  movej([1.2951, -1.388, 1.6, -0.4, 1.57, 0.0], a=1.7, v=2.0, r=0.08)
  movej([1.2954, -1.3912, 1.6, -0.4, 1.57, 0.0], a=1.7, v=2.0, r=0.08)
  movej([1.2958, -1.3945, 1.6, -0.4, 1.57, 0.0], a=1.7, v=2.0, r=0.08)
  movej([1.2961, -1.3977, 1.6, -0.4, 1.57, 0.0], a=1.7, v=2.0, r=0.08)
  movej([1.2965, -1.4009, 1.6, -0.4, 1.57, 0.0], a=1.7, v=2.0, r=0.08)
  movej([1.2969, -1.4041, 1.6, -0.4, 1.57, 0.0], a=1.7, v=2.0, r=0.08)
  movej([1.2973, -1.4072, 1.6, -0.4, 1.57, 0.0], a=1.7, v=2.0, r=0.08)
  movej([1.2977, -1.4104, 1.6, -0.4, 1.57, 0.0], a=1.7, v=2.0, r=0.08)
  movej([1.2982, -1.4135, 1.6, -0.4, 1.57, 0.0], a=1.7, v=2.0, r=0.08)
  movej([1.2986, -1.4166, 1.6, -0.4, 1.57, 0.0], a=1.7, v=2.0, r=0.08)
  movej([1.2991, -1.4196, 1.6, -0.4, 1.57, 0.0], a=1.7, v=2.0, r=0.08)
  movej([1.2996, -1.4227, 1.6, -0.4, 1.57, 0.0], a=1.7, v=2.0, r=0.08)
  movej([1.3001, -1.4257, 1.6, -0.4, 1.57, 0.0], a=1.7, v=2.0, r=0.08)
  movej([1.3006, -1.4287, 1.6, -0.4, 1.57, 0.0], a=1.7, v=2.0, r=0.08)
  movej([1.3012, -1.4317, 1.6, -0.4, 1.57, 0.0], a=1.7, v=2.0, r=0.08)
  movej([1.3018, -1.4347, 1.6, -0.4, 1.57, 0.0], a=1.7, v=2.0, r=0.08)
  movej([1.3023, -1.4376, 1.6, -0.4, 1.57, 0.0], a=1.7, v=2.0, r=0.08)
  movej([1.3029, -1.4405, 1.6, -0.4, 1.57, 0.0], a=1.7, v=2.0, r=0.08)
  movej([1.3035, -1.4433, 1.6, -0.4, 1.57, 0.0], a=1.7, v=2.0, r=0.08)
  movej([1.3042, -1.4462, 1.6, -0.4, 1.57, 0.0], a=1.7, v=2.0, r=0.08)
  movej([1.3048, -1.449, 1.6, -0.4, 1.57, 0.0], a=1.7, v=2.0, r=0.08)
  movej([1.3055, -1.4518, 1.6, -0.4, 1.57, 0.0], a=1.7, v=2.0, r=0.08)
  movej([1.3061, -1.4545, 1.6, -0.4, 1.57, 0.0], a=1.7, v=2.0, r=0.08)
  movej([1.3068, -1.4572, 1.6, -0.4, 1.57, 0.0], a=1.7, v=2.0, r=0.08)
  movej([1.3075, -1.4599, 1.6, -0.4, 1.57, 0.0], a=1.7, v=2.0, r=0.08)
  movej([1.3083, -1.4626, 1.6, -0.4, 1.57, 0.0], a=1.7, v=2.0, r=0.08)
  movej([1.309, -1.4652, 1.6, -0.4, 1.57, 0.0], a=1.7, v=2.0, r=0.08)
  movej([1.3098, -1.4678, 1.6, -0.4, 1.57, 0.0], a=1.7, v=2.0, r=0.08)
  movej([1.3105, -1.4703, 1.6, -0.4, 1.57, 0.0], a=1.7, v=2.0, r=0.08)
  movej([1.3113, -1.4728, 1.6, -0.4, 1.57, 0.0], a=1.7, v=2.0, r=0.08)
  movej([1.3121, -1.4753, 1.6, -0.4, 1.57, 0.0], a=1.7, v=2.0, r=0.08)
  movej([1.313, -1.4777, 1.6, -0.4, 1.57, 0.0], a=1.7, v=2.0, r=0.08)
  movej([1.3138, -1.4801, 1.6, -0.4, 1.57, 0.0], a=1.7, v=2.0, r=0.08)
  movej([1.3146, -1.4825, 1.6, -0.4, 1.57, 0.0], a=1.7, v=2.0, r=0.08)
  movej([1.3155, -1.4848, 1.6, -0.4, 1.57, 0.0], a=1.7, v=2.0, r=0.08)
  movej([1.3164, -1.4871, 1.6, -0.4, 1.57, 0.0], a=1.7, v=2.0, r=0.08)
  movej([1.3173, -1.4894, 1.6, -0.4, 1.57, 0.0], a=1.7, v=2.0, r=0.08)
  movej([1.3182, -1.4916, 1.6, -0.4, 1.57, 0.0], a=1.7, v=2.0, r=0.08)
  movej([1.3191, -1.4937, 1.6, -0.4, 1.57, 0.0], a=1.7, v=2.0, r=0.08)
  movej([1.3201, -1.4959, 1.6, -0.4, 1.57, 0.0], a=1.7, v=2.0, r=0.08)
  movej([1.321, -1.4979, 1.6, -0.4, 1.57, 0.0], a=1.7, v=2.0, r=0.08)
  movej([1.322, -1.5, 1.6, -0.4, 1.57, 0.0], a=1.7, v=2.0, r=0.08)
  movej([1.323, -1.502, 1.6, -0.4, 1.57, 0.0], a=1.7, v=2.0, r=0.08)
  movej([1.324, -1.5039, 1.6, -0.4, 1.57, 0.0], a=1.7, v=2.0, r=0.08)
  movej([1.3251, -1.5058, 1.6, -0.4, 1.57, 0.0], a=1.7, v=2.0, r=0.08)
  movej([1.3261, -1.5077, 1.6, -0.4, 1.57, 0.0], a=1.7, v=2.0, r=0.08)
  movej([1.3271, -1.5095, 1.6, -0.4, 1.57, 0.0], a=1.7, v=2.0, r=0.08)
  movej([1.3282, -1.5113, 1.6, -0.4, 1.57, 0.0], a=1.7, v=2.0, r=0.08)
  movej([1.3293, -1.513, 1.6, -0.4, 1.57, 0.0], a=1.7, v=2.0, r=0.08)
  movej([1.3304, -1.5147, 1.6, -0.4, 1.57, 0.0], a=1.7, v=2.0, r=0.08)
  movej([1.3315, -1.5163, 1.6, -0.4, 1.57, 0.0], a=1.7, v=2.0, r=0.08)
  movej([1.3326, -1.5179, 1.6, -0.4, 1.57, 0.0], a=1.7, v=2.0, r=0.08)
  movej([1.3338, -1.5194, 1.6, -0.4, 1.57, 0.0], a=1.7, v=2.0, r=0.08)
  movej([1.3349, -1.5209, 1.6, -0.4, 1.57, 0.0], a=1.7, v=2.0, r=0.08)
  movej([1.3361, -1.5224, 1.6, -0.4, 1.57, 0.0], a=1.7, v=2.0, r=0.08)
  movej([1.3373, -1.5238, 1.6, -0.4, 1.57, 0.0], a=1.7, v=2.0, r=0.08)
  movej([1.3385, -1.5251, 1.6, -0.4, 1.57, 0.0], a=1.7, v=2.0, r=0.08)
  movej([1.3397, -1.5264, 1.6, -0.4, 1.57, 0.0], a=1.7, v=2.0, r=0.08)
  movej([1.3409, -1.5277, 1.6, -0.4, 1.57, 0.0], a=1.7, v=2.0, r=0.08)
  movej([1.3422, -1.5288, 1.6, -0.4, 1.57, 0.0], a=1.7, v=2.0, r=0.08)
  movej([1.3434, -1.53, 1.6, -0.4, 1.57, 0.0], a=1.7, v=2.0, r=0.08)
  movej([1.3447, -1.5311, 1.6, -0.4, 1.57, 0.0], a=1.7, v=2.0, r=0.08)
  movej([1.346, -1.5321, 1.6, -0.4, 1.57, 0.0], a=1.7, v=2.0, r=0.08)
  movej([1.3473, -1.5331, 1.6, -0.4, 1.57, 0.0], a=1.7, v=2.0, r=0.08)
  movej([1.3486, -1.5341, 1.6, -0.4, 1.57, 0.0], a=1.7, v=2.0, r=0.08)
  movej([1.3499, -1.535, 1.6, -0.4, 1.57, 0.0], a=1.7, v=2.0, r=0.08)
  movej([1.3513, -1.5358, 1.6, -0.4, 1.57, 0.0], a=1.7, v=2.0, r=0.08)
  movej([1.3526, -1.5366, 1.6, -0.4, 1.57, 0.0], a=1.7, v=2.0, r=0.08)
  movej([1.354, -1.5373, 1.6, -0.4, 1.57, 0.0], a=1.7, v=2.0, r=0.08)
  movej([1.3554, -1.538, 1.6, -0.4, 1.57, 0.0], a=1.7, v=2.0, r=0.08)
  movej([1.3568, -1.5386, 1.6, -0.4, 1.57, 0.0], a=1.7, v=2.0, r=0.08)
  movej([1.3582, -1.5392, 1.6, -0.4, 1.57, 0.0], a=1.7, v=2.0, r=0.08)
  movej([1.3596, -1.5397, 1.6, -0.4, 1.57, 0.0], a=1.7, v=2.0, r=0.08)
  movej([1.361, -1.5402, 1.6, -0.4, 1.57, 0.0], a=1.7, v=2.0, r=0.08)
  movej([1.3625, -1.5406, 1.6, -0.4, 1.57, 0.0], a=1.7, v=2.0, r=0.08)
  movej([1.3639, -1.541, 1.6, -0.4, 1.57, 0.0], a=1.7, v=2.0, r=0.08)
  movej([1.3654, -1.5413, 1.6, -0.4, 1.57, 0.0], a=1.7, v=2.0, r=0.08)
  movej([1.3669, -1.5416, 1.6, -0.4, 1.57, 0.0], a=1.7, v=2.0, r=0.08)
  movej([1.3684, -1.5418, 1.6, -0.4, 1.57, 0.0], a=1.7, v=2.0, r=0.08)
  movej([1.3699, -1.5419, 1.6, -0.4, 1.57, 0.0], a=1.7, v=2.0, r=0.08)
  movej([1.3714, -1.542, 1.6, -0.4, 1.57, 0.0], a=1.7, v=2.0, r=0.08)
  movej([1.373, -1.5421, 1.6, -0.4, 1.57, 0.0], a=1.7, v=2.0, r=0.08)
  movej([1.3745, -1.5421, 1.6, -0.4, 1.57, 0.0], a=1.7, v=2.0, r=0.08)
  movej([1.3761, -1.542, 1.6, -0.4, 1.57, 0.0], a=1.7, v=2.0, r=0.08)
  movej([1.3776, -1.5419, 1.6, -0.4, 1.57, 0.0], a=1.7, v=2.0, r=0.08)
  movej([1.3792, -1.5417, 1.6, -0.4, 1.57, 0.0], a=1.7, v=2.0, r=0.08)
  movej([1.3808, -1.5415, 1.6, -0.4, 1.57, 0.0], a=1.7, v=2.0, r=0.08)
  movej([1.3824, -1.5412, 1.6, -0.4, 1.57, 0.0], a=1.7, v=2.0, r=0.08)
  movej([1.384, -1.5409, 1.6, -0.4, 1.57, 0.0], a=1.7, v=2.0, r=0.08)
  movej([1.3857, -1.5405, 1.6, -0.4, 1.57, 0.0], a=1.7, v=2.0, r=0.08)
  movej([1.3873, -1.5401, 1.6, -0.4, 1.57, 0.0], a=1.7, v=2.0, r=0.08)
  movej([1.389, -1.5396, 1.6, -0.4, 1.57, 0.0], a=1.7, v=2.0, r=0.08)
  movej([1.3906, -1.5391, 1.6, -0.4, 1.57, 0.0], a=1.7, v=2.0, r=0.08)
  movej([1.3923, -1.5385, 1.6, -0.4, 1.57, 0.0], a=1.7, v=2.0, r=0.08)
  movej([1.394, -1.5378, 1.6, -0.4, 1.57, 0.0], a=1.7, v=2.0, r=0.08)
  movej([1.3957, -1.5371, 1.6, -0.4, 1.57, 0.0], a=1.7, v=2.0, r=0.08)
  movej([1.3974, -1.5364, 1.6, -0.4, 1.57, 0.0], a=1.7, v=2.0, r=0.08)
  movej([1.3991, -1.5356, 1.6, -0.4, 1.57, 0.0], a=1.7, v=2.0, r=0.08)
  movej([1.4008, -1.5347, 1.6, -0.4, 1.57, 0.0], a=1.7, v=2.0, r=0.08)
  movej([1.4026, -1.5338, 1.6, -0.4, 1.57, 0.0], a=1.7, v=2.0, r=0.08)
  movej([1.4043, -1.5329, 1.6, -0.4, 1.57, 0.0], a=1.7, v=2.0, r=0.08)
  movej([1.4061, -1.5319, 1.6, -0.4, 1.57, 0.0], a=1.7, v=2.0, r=0.08)
  movej([1.4078, -1.5308, 1.6, -0.4, 1.57, 0.0], a=1.7, v=2.0, r=0.08)
  movej([1.4096, -1.5297, 1.6, -0.4, 1.57, 0.0], a=1.7, v=2.0, r=0.08)
  movej([1.4114, -1.5286, 1.6, -0.4, 1.57, 0.0], a=1.7, v=2.0, r=0.08)
  movej([1.4132, -1.5273, 1.6, -0.4, 1.57, 0.0], a=1.7, v=2.0, r=0.08)
  movej([1.415, -1.5261, 1.6, -0.4, 1.57, 0.0], a=1.7, v=2.0, r=0.08)
  movej([1.4168, -1.5248, 1.6, -0.4, 1.57, 0.0], a=1.7, v=2.0, r=0.08)
  movej([1.4187, -1.5234, 1.6, -0.4, 1.57, 0.0], a=1.7, v=2.0, r=0.08)
  movej([1.4205, -1.522, 1.6, -0.4, 1.57, 0.0], a=1.7, v=2.0, r=0.08)
  movej([1.4223, -1.5206, 1.6, -0.4, 1.57, 0.0], a=1.7, v=2.0, r=0.08)
  movej([1.4242, -1.5191, 1.6, -0.4, 1.57, 0.0], a=1.7, v=2.0, r=0.08)
  movej([1.4261, -1.5175, 1.6, -0.4, 1.57, 0.0], a=1.7, v=2.0, r=0.08)
  movej([1.4279, -1.5159, 1.6, -0.4, 1.57, 0.0], a=1.7, v=2.0, r=0.08)
  movej([1.4298, -1.5143, 1.6, -0.4, 1.57, 0.0], a=1.7, v=2.0, r=0.08)
  movej([1.4317, -1.5126, 1.6, -0.4, 1.57, 0.0], a=1.7, v=2.0, r=0.08)
  movej([1.4336, -1.5108, 1.6, -0.4, 1.57, 0.0], a=1.7, v=2.0, r=0.08)
  movej([1.4355, -1.509, 1.6, -0.4, 1.57, 0.0], a=1.7, v=2.0, r=0.08)
  movej([1.4374, -1.5072, 1.6, -0.4, 1.57, 0.0], a=1.7, v=2.0, r=0.08)
  movej([1.4394, -1.5053, 1.6, -0.4, 1.57, 0.0], a=1.7, v=2.0, r=0.08)
  movej([1.4413, -1.5034, 1.6, -0.4, 1.57, 0.0], a=1.7, v=2.0, r=0.08)
  movej([1.4432, -1.5015, 1.6, -0.4, 1.57, 0.0], a=1.7, v=2.0, r=0.08)
  movej([1.4452, -1.4995, 1.6, -0.4, 1.57, 0.0], a=1.7, v=2.0, r=0.08)
  movej([1.4471, -1.4974, 1.6, -0.4, 1.57, 0.0], a=1.7, v=2.0, r=0.08)
  movej([1.4491, -1.4953, 1.6, -0.4, 1.57, 0.0], a=1.7, v=2.0, r=0.08)
  movej([1.4511, -1.4932, 1.6, -0.4, 1.57, 0.0], a=1.7, v=2.0, r=0.08)
  movej([1.453, -1.491, 1.6, -0.4, 1.57, 0.0], a=1.7, v=2.0, r=0.08)
  movej([1.455, -1.4888, 1.6, -0.4, 1.57, 0.0], a=1.7, v=2.0, r=0.08)
  movej([1.457, -1.4865, 1.6, -0.4, 1.57, 0.0], a=1.7, v=2.0, r=0.08)
  movej([1.459, -1.4843, 1.6, -0.4, 1.57, 0.0], a=1.7, v=2.0, r=0.08)
  movej([1.461, -1.4819, 1.6, -0.4, 1.57, 0.0], a=1.7, v=2.0, r=0.08)
  movej([1.463, -1.4795, 1.6, -0.4, 1.57, 0.0], a=1.7, v=2.0, r=0.08)
  movej([1.4651, -1.4771, 1.6, -0.4, 1.57, 0.0], a=1.7, v=2.0, r=0.08)
  movej([1.4671, -1.4747, 1.6, -0.4, 1.57, 0.0], a=1.7, v=2.0, r=0.08)
  movej([1.4691, -1.4722, 1.6, -0.4, 1.57, 0.0], a=1.7, v=2.0, r=0.08)
  movej([1.4712, -1.4697, 1.6, -0.4, 1.57, 0.0], a=1.7, v=2.0, r=0.08)
  movej([1.4732, -1.4671, 1.6, -0.4, 1.57, 0.0], a=1.7, v=2.0, r=0.08)
  movej([1.4753, -1.4645, 1.6, -0.4, 1.57, 0.0], a=1.7, v=2.0, r=0.08)
  movej([1.4773, -1.4619, 1.6, -0.4, 1.57, 0.0], a=1.7, v=2.0, r=0.08)
  movej([1.4794, -1.4593, 1.6, -0.4, 1.57, 0.0], a=1.7, v=2.0, r=0.08)
  movej([1.4814, -1.4566, 1.6, -0.4, 1.57, 0.0], a=1.7, v=2.0, r=0.08)
  movej([1.4835, -1.4538, 1.6, -0.4, 1.57, 0.0], a=1.7, v=2.0, r=0.08)
  movej([1.4856, -1.4511, 1.6, -0.4, 1.57, 0.0], a=1.7, v=2.0, r=0.08)
  movej([1.4877, -1.4483, 1.6, -0.4, 1.57, 0.0], a=1.7, v=2.0, r=0.08)
  movej([1.4898, -1.4455, 1.6, -0.4, 1.57, 0.0], a=1.7, v=2.0, r=0.08)
  movej([1.4919, -1.4426, 1.6, -0.4, 1.57, 0.0], a=1.7, v=2.0, r=0.08)
  movej([1.494, -1.4398, 1.6, -0.4, 1.57, 0.0], a=1.7, v=2.0, r=0.08)
  movej([1.4961, -1.4369, 1.6, -0.4, 1.57, 0.0], a=1.7, v=2.0, r=0.08)
  movej([1.4982, -1.4339, 1.6, -0.4, 1.57, 0.0], a=1.7, v=2.0, r=0.08)
  movej([1.5003, -1.431, 1.6, -0.4, 1.57, 0.0], a=1.7, v=2.0, r=0.08)
  movej([1.5024, -1.428, 1.6, -0.4, 1.57, 0.0], a=1.7, v=2.0, r=0.08)
  movej([1.5045, -1.425, 1.6, -0.4, 1.57, 0.0], a=1.7, v=2.0, r=0.08)
  movej([1.5067, -1.4219, 1.6, -0.4, 1.57, 0.0], a=1.7, v=2.0, r=0.08)
  movej([1.5088, -1.4189, 1.6, -0.4, 1.57, 0.0], a=1.7, v=2.0, r=0.08)
  movej([1.5109, -1.4158, 1.6, -0.4, 1.57, 0.0], a=1.7, v=2.0, r=0.08)
  movej([1.5131, -1.4127, 1.6, -0.4, 1.57, 0.0], a=1.7, v=2.0, r=0.08)
  movej([1.5152, -1.4096, 1.6, -0.4, 1.57, 0.0], a=1.7, v=2.0, r=0.08)
  movej([1.5173, -1.4064, 1.6, -0.4, 1.57, 0.0], a=1.7, v=2.0, r=0.08)
  movej([1.5195, -1.4033, 1.6, -0.4, 1.57, 0.0], a=1.7, v=2.0, r=0.08)
  movej([1.5216, -1.4001, 1.6, -0.4, 1.57, 0.0], a=1.7, v=2.0, r=0.08)
  movej([1.5238, -1.3969, 1.6, -0.4, 1.57, 0.0], a=1.7, v=2.0, r=0.08)
  movej([1.5259, -1.3937, 1.6, -0.4, 1.57, 0.0], a=1.7, v=2.0, r=0.08)
  movej([1.5281, -1.3904, 1.6, -0.4, 1.57, 0.0], a=1.7, v=2.0, r=0.08)
  movej([1.5303, -1.3872, 1.6, -0.4, 1.57, 0.0], a=1.7, v=2.0, r=0.08)
  movej([1.5324, -1.3839, 1.6, -0.4, 1.57, 0.0], a=1.7, v=2.0, r=0.08)
  movej([1.5346, -1.3806, 1.6, -0.4, 1.57, 0.0], a=1.7, v=2.0, r=0.08)
  movej([1.5368, -1.3773, 1.6, -0.4, 1.57, 0.0], a=1.7, v=2.0, r=0.08)
  movej([1.5389, -1.374, 1.6, -0.4, 1.57, 0.0], a=1.7, v=2.0, r=0.08)
  movej([1.5411, -1.3707, 1.6, -0.4, 1.57, 0.0], a=1.7, v=2.0, r=0.08)
  movej([1.5433, -1.3674, 1.6, -0.4, 1.57, 0.0], a=1.7, v=2.0, r=0.08)
  movej([1.5454, -1.364, 1.6, -0.4, 1.57, 0.0], a=1.7, v=2.0, r=0.08)
  movej([1.5476, -1.3607, 1.6, -0.4, 1.57, 0.0], a=1.7, v=2.0, r=0.08)
  movej([1.5498, -1.3573, 1.6, -0.4, 1.57, 0.0], a=1.7, v=2.0, r=0.08)
  movej([1.552, -1.354, 1.6, -0.4, 1.57, 0.0], a=1.7, v=2.0, r=0.08)
  movej([1.5542, -1.3506, 1.6, -0.4, 1.57, 0.0], a=1.7, v=2.0, r=0.08)
  movej([1.5563, -1.3472, 1.6, -0.4, 1.57, 0.0], a=1.7, v=2.0, r=0.08)
  movej([1.5585, -1.3438, 1.6, -0.4, 1.57, 0.0], a=1.7, v=2.0, r=0.08)
  movej([1.5607, -1.3404, 1.6, -0.4, 1.57, 0.0], a=1.7, v=2.0, r=0.08)
  movej([1.5629, -1.337, 1.6, -0.4, 1.57, 0.0], a=1.7, v=2.0, r=0.08)
  movej([1.5651, -1.3336, 1.6, -0.4, 1.57, 0.0], a=1.7, v=2.0, r=0.08)
  movej([1.5673, -1.3302, 1.6, -0.4, 1.57, 0.0], a=1.7, v=2.0, r=0.08)
  movej([1.5695, -1.3268, 1.6, -0.4, 1.57, 0.0], a=1.7, v=2.0, r=0.08)
  movej([1.5716, -1.3235, 1.6, -0.4, 1.57, 0.0], a=1.7, v=2.0, r=0.08)
  movej([1.5738, -1.3201, 1.6, -0.4, 1.57, 0.0], a=1.7, v=2.0, r=0.08)
  movej([1.576, -1.3167, 1.6, -0.4, 1.57, 0.0], a=1.7, v=2.0, r=0.08)
  movej([1.5782, -1.3133, 1.6, -0.4, 1.57, 0.0], a=1.7, v=2.0, r=0.08)
  movej([1.5804, -1.3099, 1.6, -0.4, 1.57, 0.0], a=1.7, v=2.0, r=0.08)
  movej([1.5826, -1.3065, 1.6, -0.4, 1.57, 0.0], a=1.7, v=2.0, r=0.08)
  movej([1.5847, -1.3031, 1.6, -0.4, 1.57, 0.0], a=1.7, v=2.0, r=0.08)
  movej([1.5869, -1.2997, 1.6, -0.4, 1.57, 0.0], a=1.7, v=2.0, r=0.08)
  movej([1.5891, -1.2964, 1.6, -0.4, 1.57, 0.0], a=1.7, v=2.0, r=0.08)
  movej([1.5913, -1.293, 1.6, -0.4, 1.57, 0.0], a=1.7, v=2.0, r=0.08)
  movej([1.5935, -1.2896, 1.6, -0.4, 1.57, 0.0], a=1.7, v=2.0, r=0.08)
  movej([1.5956, -1.2863, 1.6, -0.4, 1.57, 0.0], a=1.7, v=2.0, r=0.08)
  movej([1.5978, -1.283, 1.6, -0.4, 1.57, 0.0], a=1.7, v=2.0, r=0.08)
  movej([1.6, -1.2796, 1.6, -0.4, 1.57, 0.0], a=1.7, v=2.0, r=0.08)
  movej([1.6022, -1.2763, 1.6, -0.4, 1.57, 0.0], a=1.7, v=2.0, r=0.08)
  movej([1.6043, -1.273, 1.6, -0.4, 1.57, 0.0], a=1.7, v=2.0, r=0.08)
  movej([1.6065, -1.2697, 1.6, -0.4, 1.57, 0.0], a=1.7, v=2.0, r=0.08)
  movej([1.6087, -1.2665, 1.6, -0.4, 1.57, 0.0], a=1.7, v=2.0, r=0.08)
  movej([1.6108, -1.2632, 1.6, -0.4, 1.57, 0.0], a=1.7, v=2.0, r=0.08)
  movej([1.613, -1.26, 1.6, -0.4, 1.57, 0.0], a=1.7, v=2.0, r=0.08)
  movej([1.6151, -1.2567, 1.6, -0.4, 1.57, 0.0], a=1.7, v=2.0, r=0.08)
  movej([1.6173, -1.2535, 1.6, -0.4, 1.57, 0.0], a=1.7, v=2.0, r=0.08)
  movej([1.6194, -1.2503, 1.6, -0.4, 1.57, 0.0], a=1.7, v=2.0, r=0.08)
  movej([1.6216, -1.2471, 1.6, -0.4, 1.57, 0.0], a=1.7, v=2.0, r=0.08)
  movej([1.6237, -1.244, 1.6, -0.4, 1.57, 0.0], a=1.7, v=2.0, r=0.08)
  movej([1.6259, -1.2409, 1.6, -0.4, 1.57, 0.0], a=1.7, v=2.0, r=0.08)
  movej([1.628, -1.2377, 1.6, -0.4, 1.57, 0.0], a=1.7, v=2.0, r=0.08)
  movej([1.6301, -1.2347, 1.6, -0.4, 1.57, 0.0], a=1.7, v=2.0, r=0.08)
  movej([1.6323, -1.2316, 1.6, -0.4, 1.57, 0.0], a=1.7, v=2.0, r=0.08)
  movej([1.6344, -1.2285, 1.6, -0.4, 1.57, 0.0], a=1.7, v=2.0, r=0.08)
  movej([1.6365, -1.2255, 1.6, -0.4, 1.57, 0.0], a=1.7, v=2.0, r=0.08)
  movej([1.6386, -1.2225, 1.6, -0.4, 1.57, 0.0], a=1.7, v=2.0, r=0.08)
  movej([1.6408, -1.2196, 1.6, -0.4, 1.57, 0.0], a=1.7, v=2.0, r=0.08)
  movej([1.6429, -1.2166, 1.6, -0.4, 1.57, 0.0], a=1.7, v=2.0, r=0.08)
  movej([1.645, -1.2137, 1.6, -0.4, 1.57, 0.0], a=1.7, v=2.0, r=0.08)
  movej([1.6471, -1.2108, 1.6, -0.4, 1.57, 0.0], a=1.7, v=2.0, r=0.08)
  movej([1.6492, -1.2079, 1.6, -0.4, 1.57, 0.0], a=1.7, v=2.0, r=0.08)
  movej([1.6513, -1.2051, 1.6, -0.4, 1.57, 0.0], a=1.7, v=2.0, r=0.08)
  movej([1.6534, -1.2023, 1.6, -0.4, 1.57, 0.0], a=1.7, v=2.0, r=0.08)
  movej([1.6554, -1.1995, 1.6, -0.4, 1.57, 0.0], a=1.7, v=2.0, r=0.08)
  movej([1.6575, -1.1968, 1.6, -0.4, 1.57, 0.0], a=1.7, v=2.0, r=0.08)
  movej([1.6596, -1.1941, 1.6, -0.4, 1.57, 0.0], a=1.7, v=2.0, r=0.08)
  movej([1.6616, -1.1914, 1.6, -0.4, 1.57, 0.0], a=1.7, v=2.0, r=0.08)
  movej([1.6637, -1.1888, 1.6, -0.4, 1.57, 0.0], a=1.7, v=2.0, r=0.08)
  movej([1.6658, -1.1862, 1.6, -0.4, 1.57, 0.0], a=1.7, v=2.0, r=0.08)
  movej([1.6678, -1.1836, 1.6, -0.4, 1.57, 0.0], a=1.7, v=2.0, r=0.08)
  movej([1.6699, -1.181, 1.6, -0.4, 1.57, 0.0], a=1.7, v=2.0, r=0.08)
  movej([1.6719, -1.1785, 1.6, -0.4, 1.57, 0.0], a=1.7, v=2.0, r=0.08)
  movej([1.6739, -1.1761, 1.6, -0.4, 1.57, 0.0], a=1.7, v=2.0, r=0.08)
  movej([1.6759, -1.1737, 1.6, -0.4, 1.57, 0.0], a=1.7, v=2.0, r=0.08)
  movej([1.678, -1.1713, 1.6, -0.4, 1.57, 0.0], a=1.7, v=2.0, r=0.08)
  movej([1.68, -1.1689, 1.6, -0.4, 1.57, 0.0], a=1.7, v=2.0, r=0.08)
  movej([1.682, -1.1666, 1.6, -0.4, 1.57, 0.0], a=1.7, v=2.0, r=0.08)
  movej([1.684, -1.1643, 1.6, -0.4, 1.57, 0.0], a=1.7, v=2.0, r=0.08)
  movej([1.686, -1.1621, 1.6, -0.4, 1.57, 0.0], a=1.7, v=2.0, r=0.08)
  movej([1.6879, -1.1599, 1.6, -0.4, 1.57, 0.0], a=1.7, v=2.0, r=0.08)
  movej([1.6899, -1.1577, 1.6, -0.4, 1.57, 0.0], a=1.7, v=2.0, r=0.08)
  movej([1.6919, -1.1556, 1.6, -0.4, 1.57, 0.0], a=1.7, v=2.0, r=0.08)
  movej([1.6938, -1.1536, 1.6, -0.4, 1.57, 0.0], a=1.7, v=2.0, r=0.08)
  movej([1.6958, -1.1515, 1.6, -0.4, 1.57, 0.0], a=1.7, v=2.0, r=0.08)
  movej([1.6977, -1.1495, 1.6, -0.4, 1.57, 0.0], a=1.7, v=2.0, r=0.08)
  movej([1.6997, -1.1476, 1.6, -0.4, 1.57, 0.0], a=1.7, v=2.0, r=0.08)
  movej([1.7016, -1.1457, 1.6, -0.4, 1.57, 0.0], a=1.7, v=2.0, r=0.08)
  movej([1.7035, -1.1439, 1.6, -0.4, 1.57, 0.0], a=1.7, v=2.0, r=0.08)
  movej([1.7054, -1.1421, 1.6, -0.4, 1.57, 0.0], a=1.7, v=2.0, r=0.08)
  movej([1.7073, -1.1403, 1.6, -0.4, 1.57, 0.0], a=1.7, v=2.0, r=0.08)
  movej([1.7092, -1.1386, 1.6, -0.4, 1.57, 0.0], a=1.7, v=2.0, r=0.08)
  movej([1.7111, -1.1369, 1.6, -0.4, 1.57, 0.0], a=1.7, v=2.0, r=0.08)
  movej([1.713, -1.1353, 1.6, -0.4, 1.57, 0.0], a=1.7, v=2.0, r=0.08)
  movej([1.7149, -1.1337, 1.6, -0.4, 1.57, 0.0], a=1.7, v=2.0, r=0.08)
  movej([1.7167, -1.1322, 1.6, -0.4, 1.57, 0.0], a=1.7, v=2.0, r=0.08)
  movej([1.7186, -1.1307, 1.6, -0.4, 1.57, 0.0], a=1.7, v=2.0, r=0.08)
  movej([1.7204, -1.1293, 1.6, -0.4, 1.57, 0.0], a=1.7, v=2.0, r=0.08)
  movej([1.7222, -1.1279, 1.6, -0.4, 1.57, 0.0], a=1.7, v=2.0, r=0.08)
  movej([1.7241, -1.1266, 1.6, -0.4, 1.57, 0.0], a=1.7, v=2.0, r=0.08)
  movej([1.7259, -1.1253, 1.6, -0.4, 1.57, 0.0], a=1.7, v=2.0, r=0.08)
  movej([1.7277, -1.124, 1.6, -0.4, 1.57, 0.0], a=1.7, v=2.0, r=0.08)
  movej([1.7295, -1.1229, 1.6, -0.4, 1.57, 0.0], a=1.7, v=2.0, r=0.08)
  movej([1.7313, -1.1217, 1.6, -0.4, 1.57, 0.0], a=1.7, v=2.0, r=0.08)
  movej([1.733, -1.1206, 1.6, -0.4, 1.57, 0.0], a=1.7, v=2.0, r=0.08)
  movej([1.7348, -1.1196, 1.6, -0.4, 1.57, 0.0], a=1.7, v=2.0, r=0.08)
  movej([1.7366, -1.1186, 1.6, -0.4, 1.57, 0.0], a=1.7, v=2.0, r=0.08)
  movej([1.7383, -1.1177, 1.6, -0.4, 1.57, 0.0], a=1.7, v=2.0, r=0.08)
  movej([1.74, -1.1168, 1.6, -0.4, 1.57, 0.0], a=1.7, v=2.0, r=0.08)
  movej([1.7418, -1.116, 1.6, -0.4, 1.57, 0.0], a=1.7, v=2.0, r=0.08)
  movej([1.7435, -1.1152, 1.6, -0.4, 1.57, 0.0], a=1.7, v=2.0, r=0.08)
  movej([1.7452, -1.1145, 1.6, -0.4, 1.57, 0.0], a=1.7, v=2.0, r=0.08)
  movej([1.7469, -1.1138, 1.6, -0.4, 1.57, 0.0], a=1.7, v=2.0, r=0.08)
  movej([1.7485, -1.1132, 1.6, -0.4, 1.57, 0.0], a=1.7, v=2.0, r=0.08)
  movej([1.7502, -1.1126, 1.6, -0.4, 1.57, 0.0], a=1.7, v=2.0, r=0.08)
  movej([1.7519, -1.1121, 1.6, -0.4, 1.57, 0.0], a=1.7, v=2.0, r=0.08)
  movej([1.7535, -1.1117, 1.6, -0.4, 1.57, 0.0], a=1.7, v=2.0, r=0.08)
  movej([1.7551, -1.1113, 1.6, -0.4, 1.57, 0.0], a=1.7, v=2.0, r=0.08)
  movej([1.7568, -1.1109, 1.6, -0.4, 1.57, 0.0], a=1.7, v=2.0, r=0.08)
  movej([1.7584, -1.1106, 1.6, -0.4, 1.57, 0.0], a=1.7, v=2.0, r=0.08)
  movej([1.76, -1.1104, 1.6, -0.4, 1.57, 0.0], a=1.7, v=2.0, r=0.08)
  movej([1.7616, -1.1102, 1.6, -0.4, 1.57, 0.0], a=1.7, v=2.0, r=0.08)
  movej([1.7631, -1.11, 1.6, -0.4, 1.57, 0.0], a=1.7, v=2.0, r=0.08)
  movej([1.7647, -1.1099, 1.6, -0.4, 1.57, 0.0], a=1.7, v=2.0, r=0.08)
  movej([1.7663, -1.1099, 1.6, -0.4, 1.57, 0.0], a=1.7, v=2.0, r=0.08)
  movej([1.7678, -1.1099, 1.6, -0.4, 1.57, 0.0], a=1.7, v=2.0, r=0.08)
  movej([1.7693, -1.11, 1.6, -0.4, 1.57, 0.0], a=1.7, v=2.0, r=0.08)
  movej([1.7708, -1.1101, 1.6, -0.4, 1.57, 0.0], a=1.7, v=2.0, r=0.08)
  movej([1.7723, -1.1103, 1.6, -0.4, 1.57, 0.0], a=1.7, v=2.0, r=0.08)
  movej([1.7738, -1.1105, 1.6, -0.4, 1.57, 0.0], a=1.7, v=2.0, r=0.08)
  movej([1.7753, -1.1108, 1.6, -0.4, 1.57, 0.0], a=1.7, v=2.0, r=0.08)
  movej([1.7768, -1.1112, 1.6, -0.4, 1.57, 0.0], a=1.7, v=2.0, r=0.08)
  movej([1.7782, -1.1116, 1.6, -0.4, 1.57, 0.0], a=1.7, v=2.0, r=0.08)
  movej([1.7797, -1.112, 1.6, -0.4, 1.57, 0.0], a=1.7, v=2.0, r=0.08)
  movej([1.7811, -1.1125, 1.6, -0.4, 1.57, 0.0], a=1.7, v=2.0, r=0.08)
  movej([1.7825, -1.1131, 1.6, -0.4, 1.57, 0.0], a=1.7, v=2.0, r=0.08)
  movej([1.7839, -1.1137, 1.6, -0.4, 1.57, 0.0], a=1.7, v=2.0, r=0.08)
  movej([1.7853, -1.1143, 1.6, -0.4, 1.57, 0.0], a=1.7, v=2.0, r=0.08)
  movej([1.7867, -1.115, 1.6, -0.4, 1.57, 0.0], a=1.7, v=2.0, r=0.08)
  movej([1.788, -1.1158, 1.6, -0.4, 1.57, 0.0], a=1.7, v=2.0, r=0.08)
  movej([1.7894, -1.1166, 1.6, -0.4, 1.57, 0.0], a=1.7, v=2.0, r=0.08)
  movej([1.7907, -1.1175, 1.6, -0.4, 1.57, 0.0], a=1.7, v=2.0, r=0.08)
  movej([1.792, -1.1184, 1.6, -0.4, 1.57, 0.0], a=1.7, v=2.0, r=0.08)
  movej([1.7933, -1.1194, 1.6, -0.4, 1.57, 0.0], a=1.7, v=2.0, r=0.08)
  movej([1.7946, -1.1204, 1.6, -0.4, 1.57, 0.0], a=1.7, v=2.0, r=0.08)
  movej([1.7959, -1.1215, 1.6, -0.4, 1.57, 0.0], a=1.7, v=2.0, r=0.08)
  movej([1.7972, -1.1226, 1.6, -0.4, 1.57, 0.0], a=1.7, v=2.0, r=0.08)
  movej([1.7984, -1.1237, 1.6, -0.4, 1.57, 0.0], a=1.7, v=2.0, r=0.08)
  movej([1.7997, -1.125, 1.6, -0.4, 1.57, 0.0], a=1.7, v=2.0, r=0.08)
  movej([1.8009, -1.1262, 1.6, -0.4, 1.57, 0.0], a=1.7, v=2.0, r=0.08)
  movej([1.8021, -1.1276, 1.6, -0.4, 1.57, 0.0], a=1.7, v=2.0, r=0.08)
  movej([1.8033, -1.1289, 1.6, -0.4, 1.57, 0.0], a=1.7, v=2.0, r=0.08)
  movej([1.8045, -1.1303, 1.6, -0.4, 1.57, 0.0], a=1.7, v=2.0, r=0.08)
  movej([1.8056, -1.1318, 1.6, -0.4, 1.57, 0.0], a=1.7, v=2.0, r=0.08)
  movej([1.8068, -1.1333, 1.6, -0.4, 1.57, 0.0], a=1.7, v=2.0, r=0.08)
  movej([1.8079, -1.1349, 1.6, -0.4, 1.57, 0.0], a=1.7, v=2.0, r=0.08)
  movej([1.809, -1.1365, 1.6, -0.4, 1.57, 0.0], a=1.7, v=2.0, r=0.08)
  movej([1.8101, -1.1382, 1.6, -0.4, 1.57, 0.0], a=1.7, v=2.0, r=0.08)
  movej([1.8112, -1.1399, 1.6, -0.4, 1.57, 0.0], a=1.7, v=2.0, r=0.08)
  movej([1.8123, -1.1416, 1.6, -0.4, 1.57, 0.0], a=1.7, v=2.0, r=0.08)
  movej([1.8134, -1.1434, 1.6, -0.4, 1.57, 0.0], a=1.7, v=2.0, r=0.08)
  movej([1.8144, -1.1452, 1.6, -0.4, 1.57, 0.0], a=1.7, v=2.0, r=0.08)
  movej([1.8155, -1.1471, 1.6, -0.4, 1.57, 0.0], a=1.7, v=2.0, r=0.08)
  movej([1.8165, -1.1491, 1.6, -0.4, 1.57, 0.0], a=1.7, v=2.0, r=0.08)
  movej([1.8175, -1.151, 1.6, -0.4, 1.57, 0.0], a=1.7, v=2.0, r=0.08)
  movej([1.8185, -1.153, 1.6, -0.4, 1.57, 0.0], a=1.7, v=2.0, r=0.08)
  movej([1.8194, -1.1551, 1.6, -0.4, 1.57, 0.0], a=1.7, v=2.0, r=0.08)
  movej([1.8204, -1.1572, 1.6, -0.4, 1.57, 0.0], a=1.7, v=2.0, r=0.08)
  movej([1.8213, -1.1593, 1.6, -0.4, 1.57, 0.0], a=1.7, v=2.0, r=0.08)
  movej([1.8222, -1.1615, 1.6, -0.4, 1.57, 0.0], a=1.7, v=2.0, r=0.08)
  movej([1.8232, -1.1638, 1.6, -0.4, 1.57, 0.0], a=1.7, v=2.0, r=0.08)
  movej([1.824, -1.166, 1.6, -0.4, 1.57, 0.0], a=1.7, v=2.0, r=0.08)
  movej([1.8249, -1.1683, 1.6, -0.4, 1.57, 0.0], a=1.7, v=2.0, r=0.08)
  movej([1.8258, -1.1707, 1.6, -0.4, 1.57, 0.0], a=1.7, v=2.0, r=0.08)
  movej([1.8266, -1.1731, 1.6, -0.4, 1.57, 0.0], a=1.7, v=2.0, r=0.08)
  movej([1.8275, -1.1755, 1.6, -0.4, 1.57, 0.0], a=1.7, v=2.0, r=0.08)
  movej([1.8283, -1.1779, 1.6, -0.4, 1.57, 0.0], a=1.7, v=2.0, r=0.08)
  movej([1.8291, -1.1804, 1.6, -0.4, 1.57, 0.0], a=1.7, v=2.0, r=0.08)
  movej([1.8298, -1.183, 1.6, -0.4, 1.57, 0.0], a=1.7, v=2.0, r=0.08)
  movej([1.8306, -1.1855, 1.6, -0.4, 1.57, 0.0], a=1.7, v=2.0, r=0.08)
  movej([1.8314, -1.1881, 1.6, -0.4, 1.57, 0.0], a=1.7, v=2.0, r=0.08)
  movej([1.8321, -1.1907, 1.6, -0.4, 1.57, 0.0], a=1.7, v=2.0, r=0.08)
  movej([1.8328, -1.1934, 1.6, -0.4, 1.57, 0.0], a=1.7, v=2.0, r=0.08)
  movej([1.8335, -1.1961, 1.6, -0.4, 1.57, 0.0], a=1.7, v=2.0, r=0.08)
  movej([1.8342, -1.1988, 1.6, -0.4, 1.57, 0.0], a=1.7, v=2.0, r=0.08)
  movej([1.8349, -1.2016, 1.6, -0.4, 1.57, 0.0], a=1.7, v=2.0, r=0.08)
  movej([1.8355, -1.2044, 1.6, -0.4, 1.57, 0.0], a=1.7, v=2.0, r=0.08)
  movej([1.8362, -1.2072, 1.6, -0.4, 1.57, 0.0], a=1.7, v=2.0, r=0.08)
  movej([1.8368, -1.2101, 1.6, -0.4, 1.57, 0.0], a=1.7, v=2.0, r=0.08)
  movej([1.8374, -1.213, 1.6, -0.4, 1.57, 0.0], a=1.7, v=2.0, r=0.08)
  movej([1.838, -1.2159, 1.6, -0.4, 1.57, 0.0], a=1.7, v=2.0, r=0.08)
  movej([1.8385, -1.2188, 1.6, -0.4, 1.57, 0.0], a=1.7, v=2.0, r=0.08)
  movej([1.8391, -1.2218, 1.6, -0.4, 1.57, 0.0], a=1.7, v=2.0, r=0.08)
  movej([1.8396, -1.2248, 1.6, -0.4, 1.57, 0.0], a=1.7, v=2.0, r=0.08)
  movej([1.8401, -1.2278, 1.6, -0.4, 1.57, 0.0], a=1.7, v=2.0, r=0.08)
  movej([1.8406, -1.2308, 1.6, -0.4, 1.57, 0.0], a=1.7, v=2.0, r=0.08)
  movej([1.8411, -1.2339, 1.6, -0.4, 1.57, 0.0], a=1.7, v=2.0, r=0.08)
  movej([1.8416, -1.237, 1.6, -0.4, 1.57, 0.0], a=1.7, v=2.0, r=0.08)
  movej([1.842, -1.2401, 1.6, -0.4, 1.57, 0.0], a=1.7, v=2.0, r=0.08)
  movej([1.8425, -1.2432, 1.6, -0.4, 1.57, 0.0], a=1.7, v=2.0, r=0.08)
  movej([1.8429, -1.2464, 1.6, -0.4, 1.57, 0.0], a=1.7, v=2.0, r=0.08)
  movej([1.8433, -1.2495, 1.6, -0.4, 1.57, 0.0], a=1.7, v=2.0, r=0.08)
  movej([1.8437, -1.2527, 1.6, -0.4, 1.57, 0.0], a=1.7, v=2.0, r=0.08)
  movej([1.844, -1.2559, 1.6, -0.4, 1.57, 0.0], a=1.7, v=2.0, r=0.08)
  movej([1.8444, -1.2591, 1.6, -0.4, 1.57, 0.0], a=1.7, v=2.0, r=0.08)
  movej([1.8447, -1.2624, 1.6, -0.4, 1.57, 0.0], a=1.7, v=2.0, r=0.08)
  movej([1.845, -1.2656, 1.6, -0.4, 1.57, 0.0], a=1.7, v=2.0, r=0.08)
  movej([1.8453, -1.2689, 1.6, -0.4, 1.57, 0.0], a=1.7, v=2.0, r=0.08)
  movej([1.8456, -1.2722, 1.6, -0.4, 1.57, 0.0], a=1.7, v=2.0, r=0.08)
  movej([1.8459, -1.2755, 1.6, -0.4, 1.57, 0.0], a=1.7, v=2.0, r=0.08)
  movej([1.8461, -1.2788, 1.6, -0.4, 1.57, 0.0], a=1.7, v=2.0, r=0.08)
  movej([1.8464, -1.2821, 1.6, -0.4, 1.57, 0.0], a=1.7, v=2.0, r=0.08)
  movej([1.8466, -1.2855, 1.6, -0.4, 1.57, 0.0], a=1.7, v=2.0, r=0.08)
  movej([1.8468, -1.2888, 1.6, -0.4, 1.57, 0.0], a=1.7, v=2.0, r=0.08)
  movej([1.847, -1.2922, 1.6, -0.4, 1.57, 0.0], a=1.7, v=2.0, r=0.08)
  movej([1.8471, -1.2955, 1.6, -0.4, 1.57, 0.0], a=1.7, v=2.0, r=0.08)
  movej([1.8473, -1.2989, 1.6, -0.4, 1.57, 0.0], a=1.7, v=2.0, r=0.08)
  movej([1.8474, -1.3023, 1.6, -0.4, 1.57, 0.0], a=1.7, v=2.0, r=0.08)
  movej([1.8475, -1.3056, 1.6, -0.4, 1.57, 0.0], a=1.7, v=2.0, r=0.08)
  movej([1.8476, -1.309, 1.6, -0.4, 1.57, 0.0], a=1.7, v=2.0, r=0.08)
  movej([1.8477, -1.3124, 1.6, -0.4, 1.57, 0.0], a=1.7, v=2.0, r=0.08)
  movej([1.8478, -1.3158, 1.6, -0.4, 1.57, 0.0], a=1.7, v=2.0, r=0.08)
  movej([1.8478, -1.3192, 1.6, -0.4, 1.57, 0.0], a=1.7, v=2.0, r=0.08)
  movej([1.8478, -1.3226, 1.6, -0.4, 1.57, 0.0], a=1.7, v=2.0, r=0.08)
  movej([1.8478, -1.326, 1.6, -0.4, 1.57, 0.0], a=1.7, v=2.0, r=0.08)
  set_tool_digital_out(0, False) # LED off — drawing done
  movej([1.57, -1.2, 1.6, -0.4, 1.57, 0.0], a=0.4, v=0.2)   # return to home
end

run_infinity_multi()
